(* PLC project Tc2_Utilities.FB_CSVMemBufferReader Demo, tc3-libraries-kb TwinCAT 3.1 *)
(* stored: creationDateTime 2026-05-11T00:00:00, modificationDateTime 2026-05-11T00:00:00 *)

PROGRAM P_Demo_FB_CSVMemBufferReader
  VAR
    fbFB_CSVMemBufferReader : FB_CSVMemBufferReader;  (* FB_CSVMemBufferReader 实例 *)
    eCmd : E_EnumCmdType := eEnumCmd_First;
    pBuffer : POINTER TO BYTE;
    cbBuffer : UDINT;
    bOk : BOOL;
    getValue : T_MaxString;
    pValue : POINTER TO BYTE;
    cbValue : UDINT;
    bCRLF : BOOL;
    cbRead : UDINT;
  END_VAR

// =============================================================================
// 场景：读配方 CSV。
// 价值：替代手写解析。
// 验证：先 Init 绑定缓冲，循环调 GetNextField 取每个字段。
// 验证步骤：
//   1. 右键 PLC 项目 → Import PLCopenXML → 选本文件
//   2. 引用 Tc2_Utilities（References → Add library）
//   3. 编译 → 登录 → 运行；按上方『验证』行的指示在线写值观察
// =============================================================================

// 单次完整调用形式（所有 VAR_INPUT 显式赋值）
fbFB_CSVMemBufferReader(
    eCmd := eCmd,
    pBuffer := pBuffer,
    cbBuffer := cbBuffer,
    bOk => bOk,
    getValue => getValue,
    pValue => pValue,
    cbValue => cbValue,
    bCRLF => bCRLF,
    cbRead => cbRead
);
END_PROGRAM
